// TIA Portal V17 export
// export: Created 2023-02-26T22:28:45.0791321Z, ExportSetting WithDefaults, DisplayName Totally Integrated Automation Portal, DisplayVersion V17, DisplayName TIA Portal Openness, DisplayVersion V17, DisplayName TIA Portal Version Control Interface, DisplayVersion V17, DisplayName TIA Portal Test Suite Advanced, DisplayVersion V17, DisplayName STEP 7 Professional, DisplayVersion V17, DisplayName SIMATIC Energy Suite, DisplayVersion V17, DisplayName STEP 7 Safety, DisplayVersion V17, DisplayName WinCC Professional, DisplayVersion V17
FUNCTION "LOG_Mode" : Void   // FC13, LAD
{ S7_Optimized_Access := 'TRUE' }
VERSION : 0.1
// stored: AutoNumber true, IsIECCheckEnabled false, SetENOAutomatically false, UDAEnableTagReadback false
BEGIN

REGION Network 1: Call: AutoControle
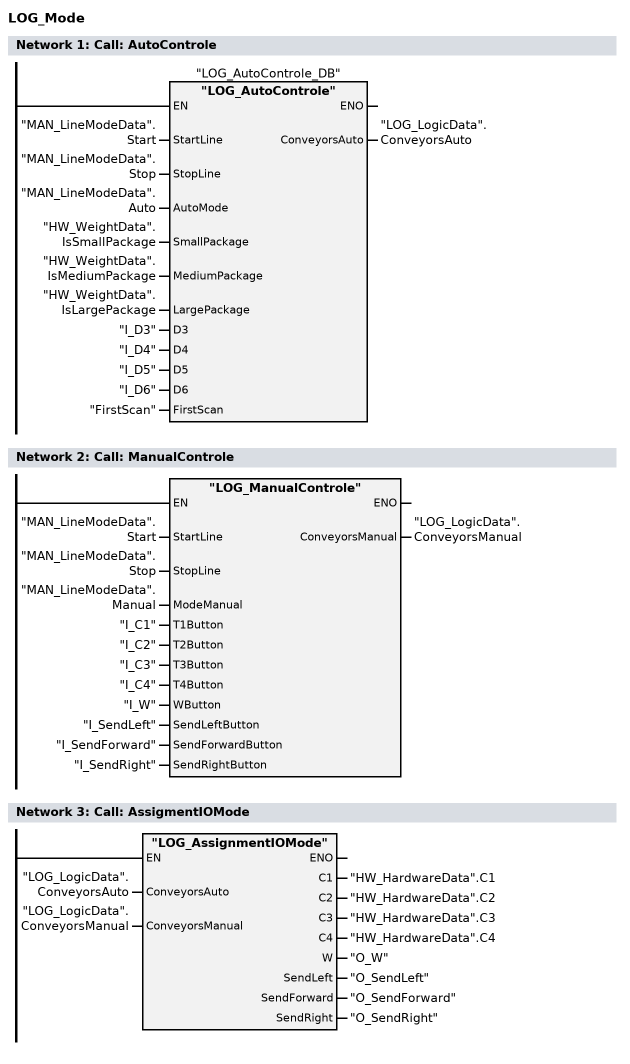
   RUNG wire#powerrail
      "LOG_AutoControle_DB"(StartLine := "MAN_LineModeData".Start, StopLine := "MAN_LineModeData".Stop, AutoMode := "MAN_LineModeData".Auto, SmallPackage := "HW_WeightData".IsSmallPackage, MediumPackage := "HW_WeightData".IsMediumPackage, LargePackage := "HW_WeightData".IsLargePackage, D3 := "I_D3", D4 := "I_D4", D5 := "I_D5", D6 := "I_D6", FirstScan := "FirstScan", ConveyorsAuto => "LOG_LogicData".ConveyorsAuto)
   END_RUNG
   // the same network as SCL:
   "LOG_AutoControle_DB"(StartLine := "MAN_LineModeData".Start,   // "LOG_AutoControle"
                         StopLine := "MAN_LineModeData".Stop,
                         AutoMode := "MAN_LineModeData".Auto,
                         SmallPackage := "HW_WeightData".IsSmallPackage,
                         MediumPackage := "HW_WeightData".IsMediumPackage,
                         LargePackage := "HW_WeightData".IsLargePackage,
                         D3 := "I_D3",
                         D4 := "I_D4",
                         D5 := "I_D5",
                         D6 := "I_D6",
                         FirstScan := "FirstScan",
                         ConveyorsAuto => "LOG_LogicData".ConveyorsAuto);
END_REGION

REGION Network 2: Call: ManualControle
   RUNG wire#powerrail
      "LOG_ManualControle"(StartLine := "MAN_LineModeData".Start, StopLine := "MAN_LineModeData".Stop, ModeManual := "MAN_LineModeData".Manual, T1Button := "I_C1", T2Button := "I_C2", T3Button := "I_C3", T4Button := "I_C4", WButton := "I_W", SendLeftButton := "I_SendLeft", SendForwardButton := "I_SendForward", SendRightButton := "I_SendRight", ConveyorsManual => "LOG_LogicData".ConveyorsManual)
   END_RUNG
   // the same network as SCL:
   "LOG_ManualControle"(StartLine := "MAN_LineModeData".Start,
                        StopLine := "MAN_LineModeData".Stop,
                        ModeManual := "MAN_LineModeData".Manual,
                        T1Button := "I_C1",
                        T2Button := "I_C2",
                        T3Button := "I_C3",
                        T4Button := "I_C4",
                        WButton := "I_W",
                        SendLeftButton := "I_SendLeft",
                        SendForwardButton := "I_SendForward",
                        SendRightButton := "I_SendRight",
                        ConveyorsManual => "LOG_LogicData".ConveyorsManual);
END_REGION

REGION Network 3: Call: AssigmentIOMode
   RUNG wire#powerrail
      "LOG_AssignmentIOMode"(ConveyorsAuto := "LOG_LogicData".ConveyorsAuto, ConveyorsManual := "LOG_LogicData".ConveyorsManual, C1 => "HW_HardwareData".C1, C2 => "HW_HardwareData".C2, C3 => "HW_HardwareData".C3, C4 => "HW_HardwareData".C4, W => "O_W", SendLeft => "O_SendLeft", SendForward => "O_SendForward", SendRight => "O_SendRight")
   END_RUNG
   // the same network as SCL:
   "LOG_AssignmentIOMode"(ConveyorsAuto := "LOG_LogicData".ConveyorsAuto,
                          ConveyorsManual := "LOG_LogicData".ConveyorsManual,
                          C1 => "HW_HardwareData".C1,
                          C2 => "HW_HardwareData".C2,
                          C3 => "HW_HardwareData".C3,
                          C4 => "HW_HardwareData".C4,
                          W => "O_W",
                          SendLeft => "O_SendLeft",
                          SendForward => "O_SendForward",
                          SendRight => "O_SendRight");
END_REGION
END_FUNCTION
